TEXTLIST TextList_ManualPage
  0 = 'GENERAL'
  1 = '1'
  2 = '2'
  3 = '3'
  4 = '4'
  5 = '5'
  6 = '6'
  7 = 'LOADING'
   = ''
END_TEXTLIST

(* stored: Version 1.1.0.1, ProductVersion 3.1.4024.12
   TextList TextList_ManualPage: Id {b8de27da-9731-42b6-b518-e2545855b80c} *)
